// TwinCAT 3 PLC project TcLog
// Title: TcLog
// Company: Benedikt Geisler
// Author: Benedikt Geisler
// ProjectVersion: 0.6.1
// Description: TcLog provides logging functionality to TwinCAT.
// ProgramVersion: 3.1.4026.20
// libraries:
//   Tc2_Standard, * (Beckhoff Automation GmbH)
//   Tc2_System, * (Beckhoff Automation GmbH)
//   Tc2_Utilities, * (Beckhoff Automation GmbH)
//   Tc3_DynamicMemory, * (Beckhoff Automation GmbH)
// project tree:
//   / Constants.TcGVL (not stored)
//   Logger/Buffer/ LogEventRingBuffer.TcPOU, LogEventBuffer.TcIO
//   Logger/Functions/ DeviceIdentification.TcPOU, FindLastOccurrence.TcPOU, GetFileExtension.TcPOU, LogLevelToAdsLogMsgType.TcPOU, RollingIntervalDetector.TcPOU, ShortenInstancePath.TcPOU, SystemTimeToNlogString.TcPOU
//   Logger/DataTypes/ Error.TcDUT, ErrorCodes.TcDUT (not stored), LogEvent.TcDUT, LoggingConfiguration.TcDUT, LogLevel.TcDUT, RollingInterval.TcDUT
//   Logger/Formatters/ DefaultAdsLogEventFormatter.TcPOU, DefaultFileLogEventFormatter.TcPOU
//   Logger/Interfaces/ ILog.TcIO (not stored), ILogCore.TcIO, LogEventFormatter.TcIO
//   Logger/TargetAdapters/ AdsLogTargetAdapter.TcPOU, FileLogTargetAdapter.TcPOU, LogTargetAdapter.TcIO
//   Logger/ TcLog.TcPOU, TcLogCore.TcPOU, TcLogTrig.TcPOU
//   StringBuilder/Interfaces/ ILimitedStringBuilder.TcIO (not stored), IStringBuilder.TcIO
//   StringBuilder/ StringBuilder.TcPOU
//   Utils/ AnyToString.TcPOU, DateTime.TcPOU, DeleteOldFiles.TcPOU (not stored), DynamicStringBuffer.TcPOU, GetFileAgeInSeconds.TcPOU
//   Utils/DataTypes/ DeleteFilesState.TcDUT, PersistToFileState.TcDUT (not stored)

// ---- Logger/DataTypes/Error.TcDUT
/// This is the error type used in this library.
TYPE Error :
STRUCT
	Active : BOOL; // `TRUE` signals an active error
	Code : INT; // Error code of type `ErrorCodes`
	Info : Tc2_System.T_MaxString; // Plain text error message
END_STRUCT
END_TYPE

// ---- Logger/DataTypes/LogEvent.TcDUT
TYPE LogEvent :
STRUCT
	timestamp : Tc2_Utilities.TimeStruct;
	level : LogLevel;
	logger : T_MaxString;
	message : T_MaxString;
END_STRUCT
END_TYPE

// ---- Logger/DataTypes/LoggingConfiguration.TcDUT
/// Configuration of TcLogCore
TYPE LoggingConfiguration :
STRUCT
	/// Whether to include the instance path of TcLog into the log message or not.
	IncludeInstancePath : BOOL;
	
	/// What is the minimum log level that gets logged?
	MinimumLevel : LogLevel;
	
	/// Which delimiter should be used between the different parts of the log string?
	Delimiter : STRING(1);
	
	/// Format of timestamp. See `TcLogCore.TimestampFormat` for formatting options.
	TimestampFormat : STRING;
	
	/// Log only valid timestamps (skip log messages during time initialization (first few cycles)
	ValidTimestampsOnly: BOOL;
END_STRUCT
END_TYPE

// ---- Logger/DataTypes/LogLevel.TcDUT
/// Log level of message to be logged.
{attribute 'qualified_only'}
{attribute 'strict'}
{attribute 'to_string'}
TYPE LogLevel :
(
	Debug := 0,
	Information,
	Warning,
	Error,
	Fatal
);
END_TYPE

// ---- Logger/DataTypes/RollingInterval.TcDUT
/// Rolling interval to create a new log file when expired. 
{attribute 'qualified_only'}
{attribute 'strict'}
{attrivute 'to_string'}
TYPE RollingInterval :
(
	None := 0,
	Hourly,
	Daily,
	Weekly,
	Monthly,
	Yearly
);
END_TYPE

// ---- Utils/DataTypes/DeleteFilesState.TcDUT
// States for state machine used in `DeleteOldFiles`.
{attribute 'qualified_only'}
{attribute 'strict'}
TYPE INTERNAL DeleteFilesState :
(
	Idle := 0,
  SearchNextFile,
  WaitUntilExecutionDone,
  ProcessFoundFiles,
  CheckIfFileIsDirectory,
  CheckFileTime,
  DeleteFile,
  FileDeleted
);
END_TYPE

// ---- Logger/Buffer/LogEventBuffer.TcIO
INTERFACE PUBLIC LogEventBuffer EXTENDS __SYSTEM.IQueryInterface

{attribute 'monitoring':='call'}
PROPERTY PUBLIC IsFull : BOOL
GET
END_GET
END_PROPERTY

METHOD PUBLIC Pop : LogEvent
END_METHOD

METHOD PUBLIC Push : BOOL
VAR_INPUT
	event : LogEvent;
END_VAR
END_METHOD

{attribute 'monitoring':='call'}
PROPERTY PUBLIC Size : UDINT
GET
END_GET
END_PROPERTY

END_INTERFACE

// ---- Logger/Interfaces/ILogCore.TcIO
INTERFACE PUBLIC ILogCore EXTENDS __SYSTEM.IQueryInterface

// Logger method.
// Logs in the standard format. This includes
// - timestamp
// - log level
// - log message
// - instance path of logging source (optional)
// The message will only be logged if the logging level exceeds the configured minimum logging level.
METHOD PUBLIC LogStandardFormat : BOOL
VAR_INPUT
	instance_path : Tc2_System.T_MaxString; // Instance path of calling logger to locate source of logging message.
	level : LogLevel; // Log level of message.
	message : Tc2_System.T_MaxString; // Data to be logged. Additional formatting wil be done.
END_VAR
END_METHOD

END_INTERFACE

// ---- Logger/Interfaces/LogEventFormatter.TcIO
INTERFACE PUBLIC LogEventFormatter EXTENDS __SYSTEM.IQueryInterface

METHOD Format : T_MaxString
VAR_INPUT
	event : LogEvent;
END_VAR
END_METHOD

END_INTERFACE

// ---- Logger/TargetAdapters/LogTargetAdapter.TcIO
INTERFACE PUBLIC LogTargetAdapter EXTENDS __System.IQueryInterface

METHOD PUBLIC Run
END_METHOD

METHOD PUBLIC SendLogEvent : BOOL
VAR_INPUT
	event : LogEvent;
END_VAR
END_METHOD

END_INTERFACE

// ---- StringBuilder/Interfaces/IStringBuilder.TcIO
{attribute 'hide'}
INTERFACE INTERNAL IStringBuilder

METHOD Append : IStringBuilder // Append text TO t current build STRING.
VAR_INPUT
    Text : Tc2_System.T_MaxString; //Text to append to current build string
END_VAR
END_METHOD

METHOD AppendIf : IStringBuilder
VAR_INPUT
    Condition : BOOL;
    Text : Tc2_System.T_MaxString;
END_VAR
END_METHOD

METHOD InsertAtLocation : IStringBuilder
VAR_INPUT
    Text : Tc2_System.T_MaxString;
    Position : INT;
END_VAR
END_METHOD

METHOD PadLeft : IStringBuilder
VAR_INPUT
    text : Tc2_System.T_MaxString; // Text to append to current build string
    length : INT; // Total length of text + padding
    c : STRING(1); // Character to be padded left of text
END_VAR
END_METHOD

METHOD Reset : ILimitedStringBuilder //Reset current build STRING TO an empty STRING.
END_METHOD

METHOD ToString : Tc2_System.T_MaxString //Returns current build STRING.
END_METHOD

END_INTERFACE

// ---- Logger/Buffer/LogEventRingBuffer.TcPOU
FUNCTION_BLOCK PUBLIC LogEventRingBuffer
VAR_GENERIC CONSTANT
	capacity : UDINT := 100;
END_VAR
IMPLEMENTS LogEventBuffer
VAR
	buffer : ARRAY[0..capacity-1] OF LogEvent;
	head : UDINT;
	tail : UDINT;
	_size : UDINT;
END_VAR

{attribute 'monitoring':='call'}
PROPERTY PUBLIC IsFull : BOOL
GET // PUBLIC
IsFull := _size = capacity;
END_GET
END_PROPERTY

METHOD PUBLIC Pop : LogEvent
VAR
	item : LogEvent;
END_VAR
IF _size = 0 THEN
	RETURN;
END_IF

item := buffer[head];
buffer[head] := 0; // Help garbage collection
head := (head + 1) MOD capacity;
_size := _size - 1;
Pop := item;
END_METHOD

METHOD PUBLIC Push : BOOL
VAR_INPUT
	item : LogEvent;
END_VAR
buffer[tail] := item;
tail := (tail + 1) MOD capacity;
IF _size < capacity THEN
	_size := _size + 1;
ELSE
	head := (head + 1) MOD capacity; // Overwrite oldest element
END_IF
END_METHOD

{attribute 'monitoring':='call'}
PROPERTY PUBLIC Size : UDINT
GET // PUBLIC
Size := _size;
END_GET
END_PROPERTY

END_FUNCTION_BLOCK

// ---- Logger/Functions/DeviceIdentification.TcPOU
FUNCTION_BLOCK DeviceIdentification
VAR
	fb : FB_GetDeviceIdentificationEx;
	initialised : BOOL;
	
	is_windows : BOOL;
	is_windows_ce : BOOL;
	is_bsd : BOOL;
	is_linux : BOOL;
	
	path_delimiter : STRING(1);
END_VAR

METHOD PUBLIC Initialise : BOOL
VAR
	dev_id : Tc2_Utilities.ST_DeviceIdentificationEx;
END_VAR
IF initialised THEN
	Initialise := initialised;
	RETURN;
END_IF

fb(bExecute := TRUE);

IF NOT fb.bBusy THEN
	dev_id := fb.stDevIdent;
	initialised := TRUE;
	fb(bExecute := FALSE);
END_IF

IF Left(dev_id.strImageOsName, 10) = 'Windows CE' THEN
	is_windows_ce := TRUE;
ELSIF Left(dev_id.strImageOsName, 7) = 'Windows' THEN
	is_windows := TRUE; 
END_IF

IF is_windows OR is_windows_ce THEN
	path_delimiter := '\';
ELSE
	path_delimiter := '/';
END_IF
END_METHOD

{attribute 'monitoring':='call'}
PROPERTY PUBLIC IsBsd : BOOL
GET // PUBLIC
IsBsd := is_bsd;
END_GET
END_PROPERTY

{attribute 'monitoring':='call'}
PROPERTY PUBLIC IsLinux : BOOL
GET // PUBLIC
IsLinux := is_linux;
END_GET
END_PROPERTY

{attribute 'monitoring':='call'}
PROPERTY PUBLIC IsWindows : BOOL
GET // PUBLIC
IsWindows := is_windows;
END_GET
END_PROPERTY

{attribute 'monitoring':='call'}
PROPERTY PUBLIC IsWindowsCE : BOOL
GET // PUBLIC
IsWindowsCE := is_windows_ce;
END_GET
END_PROPERTY

{attribute 'monitoring':='call'}
PROPERTY PUBLIC PathDelimiter : STRING(1)
GET // PUBLIC
PathDelimiter := path_delimiter;
END_GET
END_PROPERTY

END_FUNCTION_BLOCK

// ---- Logger/Functions/FindLastOccurrence.TcPOU
FUNCTION FindLastOccurrence : INT
VAR_INPUT
	within_text : T_MaxString;
	find_text : T_MaxString; 
END_VAR
VAR
	complete : BOOL;
	found_index : INT;
	new_within_text : T_MaxString;
	new_found_index : INT;
END_VAR

new_within_text := within_text;

REPEAT
	new_found_index := Find(new_within_text, find_text);
	
	IF new_found_index <> 0 THEN
		found_index := found_index + new_found_index;
		new_within_text := Right(new_within_text, Len(new_within_text) - new_found_index);
	ELSE
		complete := TRUE;
	END_IF
UNTIL complete
END_REPEAT;

FindLastOccurrence := found_index;

END_FUNCTION

// ---- Logger/Functions/GetFileExtension.TcPOU
FUNCTION GetFileExtension : T_MaxString
VAR_INPUT
	file_name : T_MaxString;
END_VAR
VAR
	last_separator_index : INT;
	extension : T_MaxString;
END_VAR

last_separator_index := FindLastOccurrence(file_name, '.');
extension := SEL(last_separator_index <> 0, '', Right(file_name, Len(file_name) - last_separator_index));
GetFileExtension := extension;

END_FUNCTION

// ---- Logger/Functions/LogLevelToAdsLogMsgType.TcPOU
// Converts TcLog.LogLevels into Tc2_System.AdsLog_MsgType.
//{attribute 'hide'}
FUNCTION INTERNAL LogLevelToAdsLogMsgType : DWORD
VAR_INPUT
  level : LogLevel;
END_VAR

CASE level OF
	LogLevel.Debug,
	LogLevel.Information:
		LogLevelToAdsLogMsgType := Tc2_System.AdsLog_MsgType_Hint;
		
	LogLevel.Warning:
		LogLevelToAdsLogMsgType := Tc2_System.AdsLog_MsgType_Warn;
		
	LogLevel.Error,
	LogLevel.Fatal:
		LogLevelToAdsLogMsgType := Tc2_System.AdsLog_MsgType_Error;
ELSE
	LogLevelToAdsLogMsgType := Tc2_System.AdsLog_MsgType_Hint;
END_CASE

END_FUNCTION

// ---- Logger/Formatters/DefaultAdsLogEventFormatter.TcPOU
{attribute 'linkalways'}
{attribute 'no_explicit_call' := 'This FB is a CLASS and must be accessed using methods or properties'}
FUNCTION_BLOCK DefaultAdsLogEventFormatter IMPLEMENTS LogEventFormatter
VAR
END_VAR

METHOD PUBLIC Format : T_MaxString
VAR_INPUT
	event : LogEvent;
END_VAR
VAR_INST
	{attribute 'hide'}
	message_builder : StringBuilder;
END_VAR
VAR CONSTANT
	DELIMITER : STRING := '|';
END_VAR
Format := message_builder
	.Reset()
	.Append(event.logger)
	.Append(DELIMITER)
	.Append(event.message)
	.ToString();
END_METHOD

END_FUNCTION_BLOCK

// ---- StringBuilder/StringBuilder.TcPOU
FUNCTION_BLOCK INTERNAL StringBuilder IMPLEMENTS IStringBuilder, ILimitedStringBuilder
VAR
  {attribute 'hide'}
  _workString : Tc2_System.T_MaxString;
END_VAR

METHOD PUBLIC Append : IStringBuilder // Append text TO t current build STRING.
VAR_INPUT
  text : Tc2_System.T_MaxString; //text to append to current build string
END_VAR
_workString:= Tc2_Standard.CONCAT(_workString,text);
Append := THIS^;
END_METHOD

METHOD PUBLIC AppendIf : IStringBuilder
VAR_INPUT
  condition : BOOL;
  text : Tc2_System.T_MaxString;
END_VAR
IF condition THEN
  _workString:= Tc2_Standard.CONCAT(_workString,text);
END_IF
AppendIf := THIS^;
END_METHOD

METHOD PUBLIC InsertAtLocation : IStringBuilder
VAR_INPUT
  text : Tc2_System.T_MaxString;
  position : INT;
END_VAR
_workString := Tc2_Standard.INSERT(_workSTring,text,position);
InsertAtLocation  := THIS^;
END_METHOD

METHOD PadLeft : IStringBuilder
VAR_INPUT
  text : Tc2_System.T_MaxString; // Text to append to current build string
  length : INT; // Total length of text + padding
  c : STRING(1); // Character to be padded left of text
END_VAR
VAR
  i : INT;
  padLength : INT;
END_VAR
// Add left padding
padLength := Tc2_Standard.LEN(text) - length;
FOR i := 1 TO padLength DO
  _workString:= Tc2_Standard.CONCAT(_workString, c);
END_FOR

// Add text
_workString:= Tc2_Standard.CONCAT(_workString,text);

PadLeft := THIS^;
END_METHOD

METHOD PUBLIC Reset : ILimitedStringBuilder //Reset current build STRING TO an empty STRING.
_workString:='';
Reset := THIS^;
END_METHOD

METHOD PUBLIC ToString : Tc2_System.T_MaxString //Returns current build STRING.
ToString := _workString;
END_METHOD

END_FUNCTION_BLOCK

// ---- Logger/Formatters/DefaultFileLogEventFormatter.TcPOU
{attribute 'linkalways'}
{attribute 'no_explicit_call' := 'This FB is a CLASS and must be accessed using methods or properties'}
FUNCTION_BLOCK DefaultFileLogEventFormatter IMPLEMENTS LogEventFormatter
VAR
END_VAR

METHOD PUBLIC Format : T_MaxString
VAR_INPUT
	event : LogEvent;
END_VAR
VAR_INST
	{attribute 'hide'}
	message_builder : StringBuilder;
END_VAR
VAR CONSTANT
	DELIMITER : STRING := '|';
END_VAR
Format := message_builder
	.Reset()
	.Append(SystemTimeToNlogString(event.timestamp))
	.Append(DELIMITER)
	.Append(TO_STRING(event.level))
	.Append(DELIMITER)
	.Append(event.logger)
	.Append(DELIMITER)
	.Append(event.message)
	.ToString();
END_METHOD

END_FUNCTION_BLOCK

// ---- Logger/Functions/SystemTimeToNlogString.TcPOU
FUNCTION INTERNAL SystemTimeToNlogString : T_MaxString
VAR_INPUT
	system_time : Tc2_Utilities.TimeStruct;
END_VAR

SystemTimeToNlogString := Tc2_Standard.Replace(Tc2_Utilities.SystemTime_To_String(system_time), ' ', 1, 11);

END_FUNCTION

// ---- Logger/Functions/RollingIntervalDetector.TcPOU
{attribute 'linkalways'}
{attribute 'no_explicit_call' := 'This FB is a CLASS and must be accessed using methods or properties'}
FUNCTION_BLOCK PUBLIC RollingIntervalDetector
VAR
	new_hour : Tc2_Standard.R_Trig;
	new_day : Tc2_Standard.R_Trig;
	new_week : Tc2_Standard.R_Trig;
	new_month : Tc2_Standard.R_Trig;
	new_year : Tc2_Standard.R_Trig;
	
	hour_rolled : BOOL;
	day_rolled : BOOL;
	week_rolled : BOOL;
	month_rolled : BOOL;
	year_rolled : BOOL;
END_VAR

PROPERTY PUBLIC DayRolled : BOOL
GET // PUBLIC
END_GET
END_PROPERTY

PROPERTY PUBLIC HourRolled : BOOL
GET // PUBLIC
END_GET
END_PROPERTY

METHOD PUBLIC IntervalRolled : BOOL
VAR_INPUT
	rolling_interval : RollingInterval;
END_VAR
CASE rolling_interval OF
	RollingInterval.Hourly:
		IntervalRolled := HourRolled;
		
	RollingInterval.Daily:
		IntervalRolled := DayRolled;
		
	RollingInterval.Weekly:
		IntervalRolled := WeekRolled;
		
	RollingInterval.Monthly:
		IntervalRolled := MonthRolled;
		
	RollingInterval.Yearly:
		IntervalRolled := YearRolled;
END_CASE
END_METHOD

PROPERTY PUBLIC MonthRolled : BOOL
GET // PUBLIC
END_GET
END_PROPERTY

METHOD PUBLIC Run
VAR_INPUT
	current_utc_time : Tc2_Utilities.TimeStruct;
END_VAR
new_hour(
	Clk := (current_utc_time.wMinute = 0 AND current_utc_time.wSecond = 0), 
	Q => hour_rolled
);

new_day(
	Clk := (hour_rolled AND current_utc_time.wHour = 0), 
	Q => day_rolled
);

new_week(
	Clk := (day_rolled AND current_utc_time.wDayOfWeek = 0),
	Q => week_rolled
);

new_month(
	Clk := (day_rolled AND current_utc_time.wDay = 1),
	Q => month_rolled
);

new_year(
	Clk := (day_rolled AND current_utc_time.wMonth = 1 AND current_utc_time.wDay = 1),
	Q => year_rolled
);
END_METHOD

PROPERTY PUBLIC WeekRolled : BOOL
GET // PUBLIC
END_GET
END_PROPERTY

PROPERTY PUBLIC YearRolled : BOOL
GET // PUBLIC
END_GET
END_PROPERTY

END_FUNCTION_BLOCK

// ---- Logger/Functions/ShortenInstancePath.TcPOU
FUNCTION INTERNAL ShortenInstancePath : T_MaxString
VAR_INPUT
	path : Tc2_System.T_MaxString; // Instance path to be shortened.
END_VAR
VAR
	i : UINT;
	shortened_path : Tc2_System.T_MaxString;
	position_in_string : INT := 0;
	position_of_last_dot : INT := 0;
END_VAR

shortened_path := path;

// Find last '.'
WHILE(Tc2_Standard.FIND(shortened_path, '.') > 0) DO
	position_in_string := Tc2_Standard.Find(shortened_path, '.');
	shortened_path := Tc2_Standard.Delete(shortened_path, position_in_string + 1, 0); 
	position_of_last_dot := position_of_last_dot + position_in_string;
END_WHILE

shortened_path := Path;

// Delete instantiation of this FB (obvious information)
shortened_path := Tc2_Standard.Delete(shortened_path, Tc2_Standard.Len(shortened_path) - position_of_last_dot + 1, position_of_last_dot);

// Delete project information
position_in_string := Tc2_Standard.Find(shortened_path, '.');
shortened_path := Tc2_Standard.Delete(shortened_path, position_in_string + 1, 0);

// Delete PLC information
position_in_string := Tc2_Standard.Find(shortened_path, '.');
shortened_path := Tc2_Standard.Delete(shortened_path, position_in_string + 1, 0);

ShortenInstancePath := shortened_path;

END_FUNCTION

// ---- Logger/TargetAdapters/AdsLogTargetAdapter.TcPOU
{attribute 'linkalways'}
{attribute 'no_explicit_call' := 'This FB is a CLASS and must be accessed using methods or properties'}
FUNCTION_BLOCK PUBLIC AdsLogTargetAdapter IMPLEMENTS LogTargetAdapter
VAR
	formatter : DefaultAdsLogEventFormatter;
END_VAR

METHOD PUBLIC Run
// Do nothing for this, as it directly logs
END_METHOD

METHOD PUBLIC SendLogEvent : BOOL
VAR_INPUT
	event : LogEvent;
END_VAR
Tc2_System.AdsLogStr(
	AdsLog_MsgType_Log OR LogLevelToAdsLogMsgType(event.level), 
	formatter.Format(event), 
	''
);
END_METHOD

END_FUNCTION_BLOCK

// ---- Logger/TargetAdapters/FileLogTargetAdapter.TcPOU
{attribute 'linkalways'}
{attribute 'no_explicit_call' := 'This FB is a CLASS and must be accessed using methods or properties'}
FUNCTION_BLOCK PUBLIC FileLogTargetAdapter IMPLEMENTS LogTargetAdapter
VAR CONSTANT
	message_buffer_capacity : UDINT := 100; // Number of messages that can be buffered
END_VAR
VAR
	// Configuration
	file_path : STRING := 'C:\';
	file_name : STRING := 'tclog.log';
	
	rolling_interval : RollingInterval := RollingInterval.Daily;
	/// When should old log files be deleted? Unit: days. Set it to `0` if log files should never be deleted. 
	log_lifespan : UINT := 0;
	timestamp_format : STRING := 'YYYYMMDD_hhmm_';

	log_cache : DynamicStringBuffer;
	date_time : DateTime;

	utc_time_as_file_time : Tc2_Utilities.T_FileTime; // Current utc time as filetime
	local_time_as_system_time : Tc2_Utilities.TimeStruct; // Current local time as timestring
	local_time_as_string : STRING; // Current local time as string

	formatter : DefaultFileLogEventFormatter;

	_error : Error; // Contains information about internal error.
	_busy : BOOL; // Logger is busy, typically with writing logs to the file system.
	
	rolling_interval_detector : RollingIntervalDetector;
	
	file_name_truncated : STRING;
	file_name_extension : STRING;
END_VAR

/// Configuration method which sets the lifespan of log files. Once exceeded, they will be deleted.
METHOD PUBLIC DeleteLogFilesAfterDays : REFERENCE TO FileLogTargetAdapter
VAR_INPUT
	/// Lifespan of logfiles in days.
	lifespan : UINT; 
END_VAR
log_lifespan := lifespan;

DeleteLogFilesAfterDays REF= THIS^;
END_METHOD

//FB_Init is always available implicitly and it is used primarily for initialization.
//The return value is not evaluated. For a specific influence, you can also declare the
//methods explicitly and provide additional code there with the standard initialization
//code. You can evaluate the return value.
METHOD FB_Init: BOOL
VAR_INPUT
    bInitRetains: BOOL; // TRUE: the retain variables are initialized (reset warm / reset cold)
    bInCopyCode: BOOL;  // TRUE: the instance will be copied to the copy code afterward (online change)   
END_VAR
log_cache.Init(message_buffer_capacity * (Tc2_System.Max_String_Length + Constants.FifoOverhead));
END_METHOD

/// Configuration method
/// Sets file_name of log file.
METHOD PUBLIC FileName : REFERENCE TO FileLogTargetAdapter
VAR_INPUT
	/// File name where the logs should be written to. Should not include path.
	file_name : STRING;
END_VAR
VAR
	last_period_index : INT;
END_VAR
THIS^.file_name := file_name;

last_period_index := FindLastOccurrence(file_name, '.');

IF last_period_index <> 0 THEN
	file_name_extension := GetFileExtension(file_name);
ELSE
	file_name_extension := 'log';
END_IF

FileName REF= THIS^;
END_METHOD

/// Configuration method
/// Sets file_path for log files.
METHOD PUBLIC FilePath : REFERENCE TO FileLogTargetAdapter
VAR_INPUT
	/// File path where the logs should be written to. Will be prefixed to `FileName`
	file_path : STRING; 
END_VAR
THIS^.file_path := file_path;

FilePath REF= THIS^;
END_METHOD

/// Flushes the logging cache. All messages that have not yet been processed will be lost.
METHOD PUBLIC FlushCache : BOOL
log_cache.FlushCache();
END_METHOD

METHOD PUBLIC Run
VAR_INST
	new_day : Tc2_Standard.R_Trig; 
	delete_expired_log_files : DeleteOldFiles;
	file_name_string_builder : StringBuilder;
	time_stamp : STRING; // Timestamp used for filename
	time_info_ready : BOOL := FALSE; // Set to true once the time information is available
	internal_error_occured : BOOL; // Aux variable to log internal errors to Error-property.
END_VAR
// Generate time data (shared state)
date_time.CyclicCall();
IF date_time.Done THEN
	time_info_ready := TRUE;
END_IF

local_time_as_system_time := date_time.AsLocalSystemTime;
local_time_as_string := date_time.AsLocalSystemTimeString;
utc_time_as_file_time := date_time.AsUtcFileTime;

rolling_interval_detector.Run(local_time_as_system_time);

// Generate new timestamp for filename
IF rolling_interval_detector.IntervalRolled(rolling_interval) OR date_time.Done THEN
	time_stamp := date_time.ToFormatString(timestamp_format);
END_IF

// Delete expired log files
new_day(Clk := local_time_as_system_time.wHour = 0);
delete_expired_log_files(
	StartScan 			:= 	new_day.Q AND (log_lifespan > 0),
	ExpirationInDays 	:=	log_lifespan,
	FilePath			:=	file_path,
	FileName 			:=	file_name,
	CurrentUtcTime 		:= 	utc_time_as_file_time	
);
IF delete_expired_log_files.Error.Active THEN
	internal_error_occured := TRUE;
	_error := delete_expired_log_files.Error;
END_IF
		
// Persist logging messages to file
log_cache.PersistToFile(
	time_info_ready,
	file_name_string_builder
		.Reset()
		.Append(file_path)
		.AppendIf(Tc2_Standard.Right(file_path, 1) <> '\', '\')
		.Append(time_stamp)
		.Append(file_name)
		.ToString()
);
IF log_cache.Error.Active THEN
	internal_error_occured := TRUE;
	_error := log_cache.Error;
END_IF

// Reset error flag each cycle to automatically confirm errors once they are gone.
IF NOT internal_error_occured THEN
	_error.Active := FALSE;
	_error.Code := ErrorCodes.None;
	_error.Info := '';
END_IF
internal_error_occured := FALSE;
END_METHOD

METHOD PUBLIC SendLogEvent : BOOL
VAR_INPUT
	event : LogEvent;
END_VAR
log_cache.AddLine(formatter.Format(event));
END_METHOD

/// Configuration method.
/// Sets the rolling interval of the log file. Once the rolling interval
/// expires, a file name with a new timestamp will be generated.
METHOD PUBLIC SetRollingInterval : REFERENCE TO FileLogTargetAdapter
VAR_INPUT
	/// Rolling interval for log file. Once exceeded, a new log file will be created.
	interval : RollingInterval; 
END_VAR
rolling_interval := interval;

SetRollingInterval REF= THIS^;
END_METHOD

END_FUNCTION_BLOCK

// ---- Logger/TcLog.TcPOU
/// `TcLog` is the client side of the logger.  
///
/// It is used to send the logs to `TcLogCore`. Typically, it is instantiated
/// once in each `FUNCTION_BLOCK` or `PROGRAM` where logging is done. The same 
/// instance can then be used for all logging within that POU. 
///
/// `TcLog` implements a string builder that facilitates the compilation of the log
/// message without the need for external data type conversions or multiple chained `CONCAT` calls.
/// See the method section for more information.
///
/// The last method to call after the log message has been built is one of ´[Debug|Information|Warning|Error|Fatal]`. 
/// This sets the log level of the message and sends it off to the log message queue of `TcLogCore` where it will
/// be processed according to its configuration.
{attribute 'linkalways'}
{attribute 'no_explicit_call' := 'This FB is a CLASS and must be accessed using methods or properties'}
//{attribute 'hide_all_locals'}
{attribute 'reflection'} 
FUNCTION_BLOCK PUBLIC TcLog IMPLEMENTS ILog
VAR
	log_condition_satisfied : BOOL; // flag that indicates, whether log condition has been satisfied.
								    // Logging will only be carried out it this evaluates to TRUE.                    
	
	log_data_initialised : BOOL; // flag that indicate, whether log data has been initialized.
							     // Necessary for configuration methods to provide a fluent interface.                            
	
	log_data : Tc2_System.T_MaxString; // contains message to be logged.
	used_logger : ILogCore;
	
	{attribute 'instance-path'} 
	{attribute 'noinit'} 
	instance_path : STRING; // contains instance path
END_VAR
VAR_STAT
	{attribute 'hide'}
	logger_singleton_instance : ILogCore; // Wires up TcLog ("Client") to TcLogCore ("Server") (Singleton-Behaviour)
END_VAR
VAR CONSTANT
	INVALID_LOGGER_REFERENCE : UDINT := 0;
END_VAR

/// Appends any given data to the log string. The type of the provided data
/// has to be one of the [standard data types](https://infosys.beckhoff.com/english.php?content=../content/1033/tc3_plc_intro/2529388939.html&id=).
/// This method can be chained.
METHOD AppendAny : REFERENCE TO TcLog
VAR_INPUT
	/// data to be appended to log string.
	data : ANY;
END_VAR
InitializeLogData();

log_data := Tc2_Standard.CONCAT(log_data, AnyToString(data));

AppendAny REF= THIS^;
END_METHOD

/// Appends a BYTE to the log string.
/// This method can be chained.
METHOD PUBLIC AppendByte : REFERENCE TO TcLog
VAR_INPUT
	/// data to be appended to log string.
	data : BYTE;
END_VAR
AppendByte REF= AppendString(TO_STRING(data));
END_METHOD

/// Appends a DATE to the log string.
/// This method can be chained.
METHOD PUBLIC AppendDate : REFERENCE TO TcLog
VAR_INPUT
  /// data to be appended to log string.
  data : DATE;
END_VAR
AppendDate REF= AppendString(TO_STRING(data));
END_METHOD

/// Appends a DATE_AND_TIME to the log string.
/// This method can be chained.
METHOD PUBLIC AppendDateAndTime : REFERENCE TO TcLog
VAR_INPUT
  /// data to be appended to log string.
  data : DATE_AND_TIME;
END_VAR
AppendDateAndTime REF= AppendString(TO_STRING(data));
END_METHOD

/// Appends a DINT to the log string.
/// This method can be chained.
METHOD PUBLIC AppendDint : REFERENCE TO TcLog
VAR_INPUT
	/// data to be appended to log string.
	data : DINT;
END_VAR
AppendDint REF= AppendString(TO_STRING(data));
END_METHOD

/// Appends a DWORD to the log string.
/// This method can be chained.
METHOD PUBLIC AppendDword : REFERENCE TO TcLog
VAR_INPUT
  /// data to be appended to log string.
  data : DWORD;
END_VAR
AppendDword REF= AppendString(TO_STRING(data));
END_METHOD

/// Appends an INT to the log string.
/// This method can be chained.
METHOD PUBLIC AppendInt : REFERENCE TO TcLog
VAR_INPUT
  /// data to be appended to log string.
  data : INT;
END_VAR
AppendInt REF= AppendString(TO_STRING(data));
END_METHOD

/// Appends a LDATE to the log string.
/// This method can be chained.
METHOD PUBLIC AppendLDate : REFERENCE TO TcLog
VAR_INPUT
  /// data to be appended to log string.
  data : LDATE;
END_VAR
AppendLDate REF= AppendString(TO_STRING(data));
END_METHOD

/// Appends a LDATE_AND_TIME to the log string.
/// This method can be chained.
METHOD PUBLIC AppendLDateAndTime : REFERENCE TO TcLog
VAR_INPUT
  /// data to be appended to log string.
  data : LDATE_AND_TIME;
END_VAR
AppendLDateAndTime REF= AppendString(TO_STRING(data));
END_METHOD

/// Appends an LINT to the log string.
/// This method can be chained.
METHOD PUBLIC AppendLint : REFERENCE TO TcLog
VAR_INPUT
  /// data to be appended to log string.
  data : LINT;
END_VAR
AppendLint REF= AppendString(TO_STRING(data));
END_METHOD

/// Appends an LREAL to the log string.
/// This method can be chained.
METHOD PUBLIC AppendLreal : REFERENCE TO TcLog
VAR_INPUT
  /// data to be appended to log string.
  data : LREAL;
END_VAR
AppendLreal REF= AppendString(TO_STRING(data));
END_METHOD

/// Appends a LTIME_OF_DAY to the log string.
/// This method can be chained.
METHOD PUBLIC AppendLTimeOfDay : REFERENCE TO TcLog
VAR_INPUT
  /// data to be appended to log string.
  data : LTIME_OF_DAY;
END_VAR
AppendLTimeOfDay REF= AppendString(TO_STRING(data));
END_METHOD

/// Appends an LWORD to the log string.
/// This method can be chained.
METHOD PUBLIC AppendLword : REFERENCE TO TcLog
VAR_INPUT
  /// data to be appended to log string.
  data : LWORD;
END_VAR
AppendLword REF= AppendString(TO_STRING(data));
END_METHOD

/// Appends a REAL to the log string.
/// This method can be chained.
METHOD PUBLIC AppendReal : REFERENCE TO TcLog
VAR_INPUT
  /// data to be appended to log string.
  data : REAL;
END_VAR
AppendReal REF= AppendString(TO_STRING(data));
END_METHOD

/// Appends a SINT to the log string.
/// This method can be chained.
METHOD PUBLIC AppendSint : REFERENCE TO TcLog
VAR_INPUT
  /// data to be appended to log string.
  data : SINT;
END_VAR
AppendSint REF= AppendString(TO_STRING(data));
END_METHOD

/// Appends another string to the log message.
/// This method can be chained.
METHOD AppendString : REFERENCE TO TcLog
VAR_INPUT
	/// data to be appended to log string.
	data : Tc2_System.T_MaxString; 
END_VAR
InitializeLogData();

log_data := Tc2_Standard.CONCAT(log_data, data);
  
AppendString REF= THIS^;
END_METHOD

/// Appends a TIME_OF_DAY to the log string.
/// This method can be chained.
METHOD PUBLIC AppendTimeOfDay : REFERENCE TO TcLog
VAR_INPUT
  /// data to be appended to log string.
  data : TIME_OF_DAY;
END_VAR
AppendTimeOfDay REF= AppendString(TO_STRING(data));
END_METHOD

/// Appends a UDINT to the log string.
/// This method can be chained.
METHOD PUBLIC AppendUdint : REFERENCE TO TcLog
VAR_INPUT
  /// data to be appended to log string.
  data : UDINT;
END_VAR
AppendUdint REF= AppendString(TO_STRING(data));
END_METHOD

/// Appends a UINT to the log string.
/// This method can be chained.
METHOD PUBLIC AppendUint : REFERENCE TO TcLog
VAR_INPUT
  /// data to be appended to log string.
  data : UINT;
END_VAR
AppendUint REF= AppendString(TO_STRING(data));
END_METHOD

/// Appends a ULINT to the log string.
/// This method can be chained.
METHOD PUBLIC AppendUlint : REFERENCE TO TcLog
VAR_INPUT
  /// data to be appended to log string.
  data : ULINT;
END_VAR
AppendUlint REF= AppendString(TO_STRING(data));
END_METHOD

/// Appends a USINT to the log string.
/// This method can be chained.
METHOD PUBLIC AppendUsint : REFERENCE TO TcLog
VAR_INPUT
  /// data to be appended to log string.
  data : USINT;
END_VAR
AppendUsint REF= AppendString(TO_STRING(data));
END_METHOD

/// Appends information about the given variable to the log string. 
/// This method can be chained.
/// Example: 

/// ```st
/// VAR
///   Logger: TcLog;
///    myInt : INT := 10;
///   myVarInfo : __SYSTEM.VAR_INFO := __VARINFO(myInt);
/// END_VAR
/// Logger.AppendVariable(myVarInfo, myInt);
/// ```
///
METHOD AppendVariable : REFERENCE TO TcLog
VAR_INPUT
	/// [VAR_INFO](https://infosys.beckhoff.com/index.php?content=../content/1031/tc3_plc_intro/3527777675.html&id=) of variable to be appended to log string.
	varInfo : __SYSTEM.VAR_INFO;
	/// Value of variable to be appended to log string.
	value : ANY; 
END_VAR
VAR
	format : Tc2_Utilities.FB_FormatString;
	symbolName : Tc2_System.T_MaxString;
	typeName : Tc2_System.T_MaxString;
END_VAR
InitializeLogData();

symbolName := varInfo.Symbol;
typeName := varInfo.TypeName; 

format(
  sFormat := '%s [%s] : ',
  arg1 := Tc2_Utilities.F_String(symbolName),
  arg2 := Tc2_Utilities.F_String(typeName));
  
AppendString(format.sOut);
AppendAny(value);

AppendVariable REF= THIS^;
END_METHOD

/// Appends a WORD to the log string.
/// This method can be chained.
METHOD PUBLIC AppendWord : REFERENCE TO TcLog
VAR_INPUT
  /// data to be appended to log string.
  data : WORD;
END_VAR
AppendWord REF= AppendString(TO_STRING(data));
END_METHOD

/// Logs the log string in DEBUG level.
METHOD PUBLIC Debug : BOOL
VAR_INPUT
	/// Message to be appended to log string.
	message : Tc2_System.T_MaxString; 
END_VAR
LogWithLevel(message, LogLevel.Debug);
END_METHOD

/// Logs the log string in ERROR level.
METHOD PUBLIC Error
VAR_INPUT
	/// Message to be appended to log string.
	message : Tc2_System.T_MaxString; 
END_VAR
LogWithLevel(message, LogLevel.Error);
END_METHOD

/// Logs the log string in FATAL level.
METHOD PUBLIC Fatal : BOOL
VAR_INPUT
	/// Message to be appended to log string.
	message : Tc2_System.T_MaxString; 
END_VAR
LogWithLevel(message, LogLevel.Fatal);
END_METHOD

/// Logs the log string in INFORMATION level.
METHOD PUBLIC Information : BOOL
VAR_INPUT
	/// Message to be appended to log string.
	message : Tc2_System.T_MaxString; 
END_VAR
LogWithLevel(message, LogLevel.Information);
END_METHOD

/// Initializes the reference to the core logger. Should only be called once from the core logger directly.
METHOD PUBLIC Init : BOOL
VAR_INPUT
	/// Reference to TcLoggerCore instance.
	log_core : ILogCore; 
END_VAR
IF logger_singleton_instance = 0 THEN
	logger_singleton_instance := log_core;
END_IF
END_METHOD

// Necessary to provide a fluent interface of the function. 
// Has to be called at the begin of any method that returns a reference to THIS^
METHOD PRIVATE InitializeLogData : BOOL
IF NOT log_data_initialised THEN
	log_condition_satisfied := TRUE;
	log_data := '';
	log_data_initialised := TRUE;
	
	IF used_logger = 0 THEN
		used_logger := logger_singleton_instance;
	END_IF
END_IF
END_METHOD

METHOD PUBLIC LogWithLevel
VAR_INPUT
	message : Tc2_System.T_MaxString;
	level : LogLevel;
END_VAR
VAR
	shortened_instance_path : T_MaxString;
	modified_message : T_MaxString;
END_VAR
InitializeLogData();

IF log_condition_satisfied THEN
	IF used_logger <> INVALID_LOGGER_REFERENCE THEN
		modified_message := Tc2_Standard.Concat(log_data, message);
 		shortened_instance_path := ShortenInstancePath(instance_path);
		used_logger.LogStandardFormat(
			shortened_instance_path,
			level,
			modified_message
		);
	ELSE
		Tc2_System.AdsLogStr(
			AdsLog_MsgType_Log OR LogLevelToAdsLogMsgType(LogLevel.Error),
			'used_logger: No valid reference',
			''
		); 
	END_IF
END_IF

log_data_initialised := FALSE;
END_METHOD

/// Conditional execution of the log command. Only executes logging when Cond = TRUE.
METHOD PUBLIC OnCondition : REFERENCE TO TcLog
VAR_INPUT
  /// Logs data only if this condition evaluates to TRUE.
  cond : BOOL; 
END_VAR
InitializeLogData();

log_condition_satisfied := cond;

OnCondition REF= THIS^;
END_METHOD

/// Initializes the reference to the core logger. This enables you to use several
/// loggers with different configurations in one project.
METHOD PUBLIC SetLogger : BOOL
VAR_INPUT
  /// Reference to Core Logger
  ref2Core : ILogCore; 
END_VAR
used_logger := ref2Core;
END_METHOD

/// Logs directly to ADS log, ignoring the settings of the base logger.
METHOD PUBLIC ToAdsLog : BOOL
VAR_INPUT
  /// Log level in which message should be logged to ADS.
  level : LogLevel; 
END_VAR
InitializeLogData();

IF log_condition_satisfied THEN
	Tc2_System.AdsLogStr(
		AdsLog_MsgType_Log OR LogLevelToAdsLogMsgType(level),
		log_data,
		''
	); 
END_IF

log_data_initialised := FALSE;
END_METHOD

/// Logs the log string in WARNING level.
METHOD PUBLIC Warning
VAR_INPUT
	/// Message to be appended to log string.
	message : Tc2_System.T_MaxString; 
END_VAR
LogWithLevel(message, LogLevel.Warning);
END_METHOD

END_FUNCTION_BLOCK

// ---- Utils/AnyToString.TcPOU
/// Converts value of input data to string, where the input type can be any of 
/// the standard data types.
FUNCTION AnyToString : Tc2_System.T_MaxString
VAR_INPUT
	/// Input data
	data : ANY;
END_VAR
VAR
	any_byte : POINTER TO BYTE;
	any_usint : POINTER TO USINT;
	_any_int : POINTER TO INT;
	any_uint : POINTER TO UINT;
	any_udint : POINTER TO UDINT;
	_anySInt : POINTER TO SINT;
	_anyDInt : POINTER TO DINT;
	_anyLInt : POINTER TO LINT;
	_anyULInt : POINTER TO ULINT;
	_anyWord : POINTER TO WORD;
	_anyLWord : POINTER TO LWORD;
	_anyReal : POINTER TO REAL;
	_anyLReal : POINTER TO LREAL;
	_anyDateAndTime : POINTER TO DATE_AND_TIME;
	_anyDate : POINTER TO DATE;
	_anyTime : POINTER TO TIME;
	_anyWString : POINTER TO WSTRING;
	_anyTOD : POINTER TO TOD;
	_anyString : POINTER TO STRING;
	_string : T_MAXSTRING;
	_wString : WSTRING;
END_VAR

IF data.TypeClass = __SYSTEM.TYPE_CLASS.TYPE_BYTE THEN
  any_byte := data.pValue;
  AnyToString := BYTE_TO_STRING(any_byte^);
    
ELSIF data.TypeClass = __SYSTEM.TYPE_CLASS.TYPE_INT THEN
  _any_int := data.pValue;
  AnyToString := INT_TO_STRING(_any_int^);
    
ELSIF data.TypeClass = __SYSTEM.TYPE_CLASS.TYPE_UINT THEN
  any_uint := data.pValue;
  AnyToString := UINT_TO_STRING(any_uint^);
    
ELSIF data.TypeClass = __SYSTEM.TYPE_CLASS.TYPE_UDINT THEN
  any_udint := data.pValue;
  AnyToString := UDINT_TO_STRING(any_udint^);
    
ELSIF data.TypeClass = __SYSTEM.TYPE_CLASS.TYPE_SINT THEN
  _anySInt := data.pValue;
  AnyToString := SINT_TO_STRING(_anySInt^);
    
ELSIF data.TypeClass = __SYSTEM.TYPE_CLASS.TYPE_USINT THEN
  any_usint := data.pValue;
  AnyToString := USINT_TO_STRING(any_usint^);
    
ELSIF data.TypeClass = __SYSTEM.TYPE_CLASS.TYPE_DINT THEN
  _anyDInt := data.pValue;
  AnyToString := DINT_TO_STRING(_anyDInt^);
    
ELSIF data.TypeClass = __SYSTEM.TYPE_CLASS.TYPE_LINT THEN
  _anyLInt := data.pValue;
  AnyToString := LINT_TO_STRING(_anyLInt^);
      
ELSIF data.TypeClass = __SYSTEM.TYPE_CLASS.TYPE_ULINT THEN
  _anyULInt := data.pValue;
  AnyToString := ULINT_TO_STRING(_anyULInt^);
  
ELSIF data.TypeClass = __SYSTEM.TYPE_CLASS.TYPE_WORD THEN
  _anyWord := data.pValue;
  AnyToString := WORD_TO_STRING(_anyWord^);
    
ELSIF data.TypeClass = __SYSTEM.TYPE_CLASS.TYPE_LWORD THEN
  _anyLWord := data.pValue;
  AnyToString := LWORD_TO_STRING(_anyLWord^);
  
ELSIF data.TypeClass = __SYSTEM.TYPE_CLASS.TYPE_REAL THEN
  _anyReal := data.pValue;
  AnyToString := REAL_TO_STRING(_anyReal^);
  
ELSIF data.TypeClass = __SYSTEM.TYPE_CLASS.TYPE_LREAL THEN
  _anyLReal := data.pValue;
  AnyToString := LREAL_TO_STRING(_anyLReal^);
  
ELSIF data.TypeClass = __SYSTEM.TYPE_CLASS.TYPE_DATEANDTIME THEN
  _anyDateAndTime := data.pValue;
  AnyToString := DT_TO_STRING(_anyDateAndTime^);  
  
ELSIF data.TypeClass = __SYSTEM.TYPE_CLASS.TYPE_DATE THEN
  _anyDate := data.pValue;
  AnyToString := DATE_TO_STRING(_anyDate^);
  
ELSIF data.TypeClass = __SYSTEM.TYPE_CLASS.TYPE_TIME THEN
  _anyTime := data.pValue;
  AnyToString := TIME_TO_STRING(_anyTime^);
  
ELSIF data.TypeClass = __SYSTEM.TYPE_CLASS.TYPE_STRING THEN
  _anyString := data.pValue;
  AnyToString := _anyString^;
  
ELSIF data.TypeClass = __SYSTEM.TYPE_CLASS.TYPE_WSTRING THEN
  _anyWString := data.pValue;
  _wString := _anyWString^;
  Tc2_Utilities.WSTRING_TO_STRING2(ADR(_string), ADR(_wString), SIZEOF(_wString));
  AnyToString := _string;
  
ELSIF data.TypeClass = __SYSTEM.TYPE_CLASS.TYPE_TIMEOFDAY THEN
  _anyTOD := data.pValue;
  AnyToString := TOD_TO_STRING(_anyTOD^);
  
ELSE
  AnyToString := TO_STRING(data.pValue^);
END_IF

END_FUNCTION

// ---- Utils/DynamicStringBuffer.TcPOU
{attribute 'no_explicit_call' := 'This FB is a CLASS and must be accessed using methods or properties'}
{attribute 'hide_all_locals'}
FUNCTION_BLOCK INTERNAL DynamicStringBuffer
VAR_OUTPUT
	Error : Error; // Error information of this FB
END_VAR
VAR
	_fifo : Tc2_Utilities.FB_StringRingBuffer; // Necessary to buffer log data until it has been written to file.
	_memoryManager : Tc3_DynamicMemory.FB_DynMem_Manager; // Memory manager, required by DynMem_Buffer.
	_dynamicMemoryBuffer : Tc3_DynamicMemory.FB_DynMem_Buffer(ipMemMan := _memoryManager); // Provides dynamic buffer for Fifo. Is extended automatically if more than the
																   // default buffer size is needed.                  
	_busy : BOOL; // Buffer is busy; typically with writing data to the file system.
END_VAR

METHOD AddLine : BOOL
VAR_INPUT
  text : Tc2_System.T_MaxString; // Text to be added to the buffer
END_VAR
ResizeFifoBufferIfNecessary();
_fifo.A_AddTail(putValue := Tc2_Standard.CONCAT(Tc2_Standard.LEFT(text, 254), '$N'));
END_METHOD

METHOD AddString : BOOL
VAR_INPUT
  text : Tc2_System.T_MaxString; // String to be added to the buffer
END_VAR
ResizeFifoBufferIfNecessary();
_fifo.A_AddTail(putValue := text);
END_METHOD

METHOD PRIVATE AllocateBuffer : BOOL // Allocates buffer FOR the fifo.
VAR_INPUT
  bufferSize : UDINT; // Initial buffer size in BYTEs for fifo buffer.
END_VAR
_dynamicMemoryBuffer.CreateBuffer(nSize:=bufferSize, bReset:=TRUE);
_fifo.pBuffer := _dynamicMemoryBuffer.pBuffer;
_fifo.cbBuffer := bufferSize;
END_METHOD

{attribute 'monitoring':='call'}
PROPERTY Busy : BOOL
GET
Busy := _busy;
END_GET
SET // PRIVATE
_busy := Busy;
END_SET
END_PROPERTY

METHOD FB_exit : BOOL
VAR_INPUT
  bInCopyCode : BOOL; // if TRUE, the exit method is called for exiting an instance that is copied afterwards (online change).
END_VAR
_dynamicMemoryBuffer.Clear();
END_METHOD

METHOD FlushCache : BOOL
_fifo.A_Reset();
END_METHOD

METHOD INTERNAL Init : BOOL
VAR_INPUT
	bufferSize : UDINT; // Initial buffer size in BYTEs for fifo buffer.
END_VAR
AllocateBuffer(bufferSize);
END_METHOD

{attribute 'hide_all_locals'}
METHOD PersistToFile : BOOL
VAR_INPUT
  enable: BOOL; // TRUE starts persistence mechanism
  fileName : Tc2_System.T_MaxString; // File name including its path
END_VAR
VAR_INST
  state : PersistToFileState;
  
  fileOpen : Tc2_System.FB_FileOpen;
  fileHandle : UINT;
  
  fileWrite : Tc2_System.FB_FileWrite;
  lockFileWriteToForceRisingEdge : BOOL; // filePuts can only be executed every other cycle
                                         // since it needs a rising edge to execute.
  fileClose : Tc2_System.FB_FileClose;
  
  buffer : ARRAY[0..CONSTANTS.BufferSize] OF BYTE;
  currentBufferPos : UDINT;
  fifoHeadString : Tc2_System.T_MaxString;
  fifoHeadLength : UDINT;
  fifoHeadBytes : ARRAY[0..Tc2_System.MAX_STRING_LENGTH] OF BYTE;
  i : UINT;
END_VAR
VAR CONSTANT
  NetId : STRING := '';
  Timeout : TIME := DEFAULT_ADS_TIMEOUT;
  MaxLogsPerCycle : UINT := UDINT_TO_UINT(CONSTANTS.BufferSize / Tc2_System.MAX_STRING_LENGTH);
  MaxBufferPosition : UDINT := (SIZEOF(buffer)-Tc2_System.MAX_STRING_LENGTH);
END_VAR
// State machine
// Using if-statements instead of case for performance reasons:
// Some states execute instantly and allow thus the next state 
// to start within the same plc cycle.

// *** I D L E ***
IF state = PersistToFileState.Idle THEN
  lockFileWriteToForceRisingEdge := FALSE;
  IF _fifo.nCount > 0 AND enable THEN 
    lockFileWriteToForceRisingEdge := FALSE;
    state := PersistToFileState.OpenFile;
  END_IF
END_IF
    
// *** O P E N   F I L E ***
fileOpen(sNetId := NetId, sPathName := fileName, nMode := FOPEN_MODEAPPEND OR FOPEN_MODETEXT, 
           ePath := PATH_GENERIC, bExecute := (state = PersistToFileState.OpenFile), tTimeout := Timeout,
           hFile => fileHandle);

IF state = PersistToFileState.OpenFile THEN
  IF fileOpen.bError THEN
    state := PersistToFileState.CloseFile;
  ELSIF NOT fileOpen.bBusy THEN
    state := PersistToFileState.GetStringFromFifo; 
  END_IF
END_IF 

// *** P O P   F R O M   F I F O ***
IF state = PersistToFileState.GetStringFromFifo THEN
  IF NOT lockFileWriteToForceRisingEdge THEN
    currentBufferPos := 0;
    FOR i:=0 TO MaxLogsPerCycle DO
      IF _fifo.nCount <= 0 THEN EXIT; END_IF
      IF currentBufferPos >= MaxBufferPosition THEN EXIT; END_IF
      
      _fifo.A_RemoveHead(getValue => fifoHeadString); 
      fifoHeadBytes := MAXSTRING_TO_BYTEARR(fifoHeadString);
      fifoHeadLength := INT_TO_UDINT(LEN(fifoHeadString));
      MEMCPY(
        destAddr  :=  ADR(buffer) + SIZEOF(BYTE) * currentBufferPos,
        srcAddr   :=  ADR(fifoHeadBytes),
        n     :=  fifoHeadLength);    
      currentBufferPos := currentBufferPos + fifoHeadLength;  
    END_FOR
    state := PersistToFileState.AppendDataToFile;
  END_IF
  lockFileWriteToForceRisingEdge := FALSE;
END_IF
  
// *** W R I T E   T O   F I L E ***
fileWrite(
  sNetId := NetId, 
  hFile := fileHandle, 
  pWriteBuff := ADR(buffer),
  cbWriteLen := currentBufferPos,
  bExecute := state = PersistToFileState.AppendDataToFile, 
  tTimeout := Timeout); 

IF state = PersistToFileState.AppendDataToFile THEN
  lockFileWriteToForceRisingEdge := TRUE;   
  IF fileWrite.bError THEN
    state := PersistToFileState.CloseFile;
  ELSIF _fifo.nCount > 0 AND NOT fileWrite.bBusy THEN
    state := PersistToFileState.GetStringFromFifo; 
  ELSIF _fifo.nCount = 0 THEN
    state := PersistToFileState.CloseFile;
  END_IF
END_IF
    
// *** C L O S E   F I L E ***
fileClose(
  sNetId := NetId, hFile := fileHandle, 
  bExecute := (state = PersistToFileState.CloseFile), tTimeout := Timeout);

IF state = PersistToFileState.CloseFile THEN
  IF NOT fileClose.bBusy THEN state := PersistToFileState.Idle; END_IF
END_IF

// Close file in case of error
IF fileOpen.bError THEN state := PersistToFileState.CloseFile; END_IF
IF fileWrite.bError THEN state := PersistToFileState.CloseFile; END_IF
IF NOT _fifo.bOk AND _fifo.nCount > 0 AND state <> PersistToFileState.Idle THEN 
  state := PersistToFileState.CloseFile; 
END_IF

// Error handling
IF fileOpen.bError THEN
  Error.Active := TRUE;
  Error.Code := ErrorCodes.OpeningFileFailed;
  Error.Info := Tc2_Standard.CONCAT('Opening file failed. Error thrown by FB_FileOpen. Consult Beckhoff InfoSys. Internal Error: ', UDINT_TO_STRING(fileOpen.nErrId));
ELSIF fileWrite.bError THEN
  Error.Active := TRUE;
  Error.Code := ErrorCodes.WritingToFileFailed;
  Error.Info := Tc2_Standard.CONCAT('Writing to file failed. Error thrown by FB_FileWrite. Consult Beckhoff InfoSys. Internal Error: ', UDINT_TO_STRING(fileWrite.nErrId));
ELSIF fileClose.bError THEN
  Error.Active := TRUE;
  Error.Code := ErrorCodes.ClosingFileFailed;
  Error.Info := Tc2_Standard.CONCAT('Closing file failed. Error thrown by FB_FileClose. Consult Beckhoff InfoSys. Internal Error: ', UDINT_TO_STRING(fileClose.nErrId));
ELSIF NOT _fifo.bOk AND _fifo.nCount > 0 THEN
  Error.Active := TRUE;
  Error.Code := ErrorCodes.FifoOverflow;
  Error.Info := 'FIFO overflow. Check if plc has enough free memory.';
ELSE
  Error.Active := FALSE;
  Error.Code := ErrorCodes.None;
  Error.Info := '';
END_IF

// Set busy state
Busy := (state <> PersistToFileState.Idle OR _fifo.nCount > 0);

(* Uncomment for cyclic logging of state machine, buffer usage & errors

ADSLOGSTR(ADSLOG_MSGTYPE_LOG, 
  Tc2_Standard.CONCAT('****DynamicStringBuffer.state:', 
  Tc2_Standard.CONCAT(UINT_TO_STRING(state),
  Tc2_Standard.CONCAT(', DynamicStringBuffer.hFile:', UINT_TO_STRING(hFile)))), '');

ADSLOGSTR(ADSLOG_MSGTYPE_LOG, 
  Tc2_Standard.CONCAT('****Fifo: used ', 
  Tc2_Standard.CONCAT(UDINT_TO_STRING(Fifo.cbSize),
  Tc2_Standard.CONCAT(' of ', UDINT_TO_STRING(Fifo.cbBuffer)))), '');
  
IF Error.Active THEN
  ADSLOGSTR(ADSLOG_MSGTYPE_LOG, 
    Tc2_Standard.CONCAT('****DynamicStringBuffer.Error: ', Error.Info), 
    '');  
END_IF
*)
END_METHOD

METHOD PopHead : Tc2_System.T_MaxString
VAR_INST
  headString : Tc2_System.T_MaxString;
END_VAR
_fifo.A_RemoveHead(getValue => headString);
PopHead := headString;
END_METHOD

// Resizes the buffer for the FIFO if necessary
METHOD PRIVATE ResizeFifoBufferIfNecessary : BOOL
VAR
  requiredSize : UDINT;
  newSize : DINT;
END_VAR
requiredSize := _fifo.cbSize + (Tc2_System.MAX_STRING_LENGTH + Constants.FifoOverhead);

IF requiredSize > _fifo.cbBuffer THEN
  _dynamicMemoryBuffer.Resize(nSize := requiredSize*SIZEOF(BYTE), bPreserve:=TRUE, bReset:=TRUE);
  _fifo.pBuffer := _dynamicMemoryBuffer.pBuffer;
  _fifo.cbBuffer := requiredSize;
END_IF
END_METHOD

END_FUNCTION_BLOCK

// ---- Utils/DateTime.TcPOU
/// Generate time data in different formats.
{attribute 'no_explicit_call' := 'This FB is a CLASS and must be accessed using methods or properties'}
{attribute: 'hide_all_locals'}
FUNCTION_BLOCK DateTime
VAR
	local_system_time : Tc2_Utilities.FB_LocalSystemTime;
	get_system_time : Tc2_System.GetSystemTime;
	time_zone_info : Tc2_Utilities.FB_GetTimeZoneInformation;
	local_time : Tc2_Utilities.FB_SystemTimeToTzSpecificLocalTime;
	local_system_time_valid : Tc2_Standard.R_Trig;
	utc_time : Tc2_Utilities.FB_TzSpecificLocalTimeToFileTime;
END_VAR

/// Returns local time as `Tc2_Utilities.T_FileTime`.
{attribute 'monitoring':='variable'}
PROPERTY AsLocalFileTime : Tc2_Utilities.T_FileTime
GET
AsLocalFileTime := SYSTEMTIME_TO_FILETIME(THIS^.AsLocalSystemTime);
END_GET
END_PROPERTY

/// Returns local time as `Tc2_Utilities.TimeStruct`.
{attribute 'monitoring':='variable'}
PROPERTY AsLocalSystemTime : Tc2_Utilities.TimeStruct
GET
AsLocalSystemTime := local_system_time.systemTime;
END_GET
END_PROPERTY

/// Returns local time as string.
{attribute 'monitoring':='variable'}
PROPERTY AsLocalSystemTimeString : Tc2_System.T_MaxString
GET
AsLocalSystemTimeString := Tc2_Utilities.SystemTime_To_String(THIS^.AsLocalSystemTime);
END_GET
END_PROPERTY

/// Returns UTC time as `Tc2_Utilities.T_FileTime`.
{attribute 'monitoring':='variable'}
PROPERTY AsUtcFileTime : Tc2_Utilities.T_FileTime
GET
AsUtcFileTime := utc_time.out;
END_GET
END_PROPERTY

METHOD CyclicCall
// Get local system time
local_system_time(
	sNetID  :=  '',
	bEnable :=  TRUE,
	dwCycle :=  1,
	dwOpt :=  1,
	tTimeout:=  DEFAULT_ADS_TIMEOUT
);

// Get timezone information
time_zone_info(
	sNetID := '',
	bExecute := TRUE,
	tTimeout := DEFAULT_ADS_TIMEOUT
);

// Convert local time to utc time
utc_time(
	in := THIS^.AsLocalFileTime,
	tzInfo := time_zone_info.tzInfo
);
 
// Finished retrieving time data
local_system_time_valid(Clk := local_system_time.bValid);
END_METHOD

/// When calling `DateTime` the first time, it takes some time until all time and timezone information is available.
/// `Done` is `TRUE` for one cycle, once all the data is ready. 
{attribute 'monitoring':='call'}
PROPERTY Done : BOOL
GET
Done := local_system_time_valid.Q;
END_GET
END_PROPERTY

// Replaces placeholders in format string by the actual time values.
{attribute 'hide_all_locals'}
{attribute 'hide'}
METHOD PRIVATE ReplaceFormatPlaceholder : STRING
VAR_INPUT
	format : STRING;
	length : INT;
	time_type : STRING(1);
END_VAR
VAR_INST
	i : INT;
	replace_string : STRING;
	time_string : STRING;
END_VAR
VAR
	local_system_time : Tc2_Utilities.TimeStruct;
END_VAR
local_system_time := THIS^.AsLocalSystemTime;

IF    time_type = 'Y' THEN time_string := TO_STRING(local_system_time.wYear);
ELSIF time_type = 'M' THEN time_string := TO_STRING(local_system_time.wMonth);
ELSIF time_type = 'D' THEN time_string := TO_STRING(local_system_time.wDay);
ELSIF time_type = 'h' THEN time_string := TO_STRING(local_system_time.wHour);
ELSIF time_type = 'm' THEN time_string := TO_STRING(local_system_time.wMinute);
ELSIF time_type = 's' THEN time_string := TO_STRING(local_system_time.wSecond);
ELSIF time_type = 'i' THEN time_string := TO_STRING(local_system_time.wMilliseconds);
ELSE
	time_string := '';
END_IF

replace_string := '';

IF length > Tc2_Standard.Len(time_string) THEN
	FOR i:=1 TO length - Tc2_Standard.Len(time_string) DO
		replace_string := Tc2_Standard.Concat(replace_string, '0');
	END_FOR
	replace_string := Tc2_Standard.Concat(replace_string, time_string);
ELSE
	replace_string := Tc2_Standard.Right(time_string, length);
END_IF

ReplaceFormatPlaceholder := Tc2_Standard.Replace(format, replace_string, length, Tc2_Standard.Find(format, time_type));
END_METHOD

/// Returns a formatted string containing the actual time information 
/// - `Y` : year
/// - `M` : month
/// - `D` : day
/// - `h` : hour 
/// - `m` : minute
/// - `s` : second
/// - `i` : millisecond
/// 
/// Example:    
/// _YYMMDD-hh:mm:ss:iii_   
/// => _20210812-12:30:22:123_
{attribute 'hide_all_locals'}
METHOD PUBLIC ToFormatString : Tc2_System.T_MaxString
VAR_INPUT
  /// Format the timestamp should have.
  format : STRING;
END_VAR
VAR_INST
  inputString : STRING;
  c : STRING(1);
  formattedString : Tc2_System.T_MaxString;
END_VAR
VAR
  year : INT := 0;
  month : INT := 0;
  day : INT := 0;
  hour : INT := 0;
  minute : INT := 0;
  second : INT := 0;
  millisecond : INT := 0;
END_VAR
VAR CONSTANT
  ValidFormat : STRING := 'YMDhms';
END_VAR
// Parses "format" and returns a adequatly formatted string containing the time information
inputString := format;

WHILE Tc2_Standard.LEN(inputString) > 0 DO
  c := Tc2_Standard.LEFT(inputString, 1);
  
  IF    c = 'Y' THEN year := year + 1;
  ELSIF c = 'M' THEN month := month + 1;
  ELSIF c = 'D' THEN day := day + 1;
  ELSIF c = 'h' THEN hour := hour + 1;
  ELSIF c = 'm' THEN minute := minute + 1;
  ELSIF c = 's' THEN second := second + 1;
  ELSIF c = 'i' THEN millisecond := millisecond + 1;
  END_IF
  
  inputString := Tc2_Standard.DELETE(inputString, 1, 1);
END_WHILE

formattedString := ReplaceFormatPlaceholder(format, year, 'Y');
formattedString := ReplaceFormatPlaceholder(formattedString, month, 'M');
formattedString := ReplaceFormatPlaceholder(formattedString, day, 'D');
formattedString := ReplaceFormatPlaceholder(formattedString, hour, 'h');
formattedString := ReplaceFormatPlaceholder(formattedString, minute, 'm');
formattedString := ReplaceFormatPlaceholder(formattedString, second, 's');
formattedString := ReplaceFormatPlaceholder(formattedString, millisecond, 'i');

ToFormatString := formattedString;
END_METHOD

END_FUNCTION_BLOCK

// ---- Logger/TcLogCore.TcPOU
/// `TcLogCore` provides the base functionality of the logger and sets the configuration.
/// The logger can be configured by calling its methods that set the configuration.
///
/// > [!NOTE]
/// > `TcLogCore.RunLogger()` should be called once each cycle. The configuration methods should be called **before** 
/// > `RunLogger` is called.
///
/// When declaring an instance of TcLogCore, the ininital buffer size has to be set. If the buffer size is set too low, it will expand
/// automatically if enough memory is available.
///
/// To set the inital buffer size to accomodate 100 messages, use it like this:
///
/// ```st
/// VAR
///   my_logger: TcLogCore(BufferSize := 100 * (Tc2_System.MAX_STRING_LENGTH * Constants.FifoOverhead));
/// END_VAR
/// ```
///
{attribute 'linkalways'}
{attribute 'no_explicit_call' := 'This FB is a CLASS and must be accessed using methods or properties'}
//{attribute 'hide_all_locals'}
FUNCTION_BLOCK PUBLIC TcLogCore IMPLEMENTS ILogCore
VAR
	logging_singleton : TcLog; // Logger-Singleton: Required to provide Singleton-functionality for TcLog.
	utc_time_as_file_time : Tc2_Utilities.T_FileTime; // Current utc time as filetime
	local_time_as_system_time : Tc2_Utilities.TimeStruct; // Current local time as timestring
	local_time_as_string : STRING; // Current local time as string
	log_cache : DynamicStringBuffer; // Dynamic string buffer to cache logs to be processed
	start_logging_configuration : BOOL; // Aux variable to provide fluent interface.
	internal_error_occured : BOOL; // Aux variable to log internal errors to Error-property.                                                   				
	_config : LoggingConfiguration := (
		MinimumLevel := LogLevel.Debug,
		Delimiter := '|',
		IncludeInstancePath := FALSE,
		TimestampFormat := 'YYYYMMDD_hhmm_',
		ValidTimestampsOnly := FALSE
	); // Logging configuration. Is set by invoking configuration methods.
	_error : Error; // Contains information about internal error.
	_busy : BOOL; // Logger is busy, typically with writing logs to the file system.
	time_info_ready : BOOL := FALSE; // Set to true once the time information is available
	
	default_log_target_adapter : AdsLogTargetAdapter;

	adapter_1 : LogTargetAdapter := default_log_target_adapter;
	adapter_2 : LogTargetAdapter;
	adapter_3 : LogTargetAdapter;
END_VAR

// Nothing to be done here. Logger works by invoking its methods.
// "RunLogger" contains all the implementation that has to be processed cyclically.

METHOD PUBLIC AddAdapter1 : REFERENCE TO TcLogCore
VAR_INPUT
	adapter : LogTargetAdapter;
END_VAR
IF adapter <> 0 THEN
	adapter_1 := adapter;
END_IF

AddAdapter1 REF= THIS^;
END_METHOD

METHOD PUBLIC AddAdapter2 : REFERENCE TO TcLogCore
VAR_INPUT
	adapter : LogTargetAdapter;
END_VAR
IF adapter <> 0 THEN
	adapter_2 := adapter;
END_IF

AddAdapter2 REF= THIS^;
END_METHOD

METHOD PUBLIC AddAdapter3 : REFERENCE TO TcLogCore
VAR_INPUT
	adapter : LogTargetAdapter;
END_VAR
IF adapter <> 0 THEN
	adapter_3 := adapter;
END_IF

AddAdapter3 REF= THIS^;
END_METHOD

/// `Busy` evaluates to `TRUE` as long as the log file is kept open to append new log messages
/// or there are pending messages in the queue to be written to the logfile.
{attribute 'monitoring':='call'}
PROPERTY PUBLIC Busy : BOOL
GET // PUBLIC
Busy := _busy;
END_GET
SET // PRIVATE
_busy := Busy;
END_SET
END_PROPERTY

/// Returns the current configuration of the logger.
{attribute 'monitoring':='variable'}
PROPERTY PUBLIC Configuration : LoggingConfiguration
GET // PUBLIC
Configuration := _config;
END_GET
END_PROPERTY

/// Returns information about internal errors.
{attribute 'monitoring':='call'}
{attribute 'suppress_wrn_C0410'}
PROPERTY Error : REFERENCE TO Error
GET
Error REF= _error;
END_GET
END_PROPERTY

METHOD FB_init : BOOL
VAR_INPUT
	bInitRetains : BOOL; // if TRUE, the retain variables are initialized (warm start / cold start)
	bInCopyCode : BOOL; // if TRUE, the instance afterwards gets moved into the copy code (online change)
	/// Initial buffer size for the internal log message buffer
	bufferSize : UDINT;
END_VAR
logging_singleton.Init(THIS^);
log_cache.Init(bufferSize);
END_METHOD

/// Configuration method. If this method is called, the instance path where the log 
/// messages has been triggered will be included in the log message. 
METHOD PUBLIC IncludeInstancePath : REFERENCE TO TcLogCore
_config.IncludeInstancePath := TRUE;

IncludeInstancePath REF= This^;
END_METHOD

/// Logger method. It should only be called from within objects that implement `ILog`.
/// Logs in the standard format. This includes
/// - timestamp
/// - log level
/// - log message
/// - instance path of logging source (optional)
/// The message will only be logged if the logging level exceeds the configured minimum logging level.
METHOD PUBLIC LogStandardFormat : BOOL
VAR_INPUT
	/// Instance path of calling logger to locate source of logging message.
	instance_path : Tc2_System.T_MaxString;

	/// Log level of message. 
	level : LogLevel; 

	/// Data to be logged.
	message : Tc2_System.T_MaxString;	
END_VAR
VAR_INST
	event : LogEvent;
END_VAR
IF level >= _config.MinimumLevel AND (TimeInfoReady OR NOT _config.ValidTimestampsOnly) THEN
	event.timestamp := local_time_as_system_time;
	event.level := level;
	event.logger := instance_path;
	event.message := message;

	IF adapter_1 <> 0 THEN
		adapter_1.SendLogEvent(event);
	END_IF
	
	IF adapter_2 <> 0 THEN
		adapter_2.SendLogEvent(event);
	END_IF
	
	IF adapter_3 <> 0 THEN
		adapter_3.SendLogEvent(event);
	END_IF
END_IF
END_METHOD

/// Configuration method.
/// Sets the minimum log level. Log messages below this level 
/// will not be logged.
METHOD PUBLIC MinimumLevel : REFERENCE TO TcLogCore
VAR_INPUT
  /// Minimum log level to be logged.
	level : LogLevel; 
END_VAR
_config.MinimumLevel := level;

MinimumLevel REF=THIS^;
END_METHOD

/// Cyclic method of Logger.
/// This method has to be executed in every PLC cycle and runs 
/// all internal methods that have to be executed cyclically.
/// > [!NOTE]
/// > This method should be the last method of `TcLogCore` to be called in each cycle.
{attribute 'hide_all_locals'}
METHOD PUBLIC RunLogger : BOOL
VAR_INST
	new_day : Tc2_Standard.R_Trig; 
	date_time : DateTime;
	delete_expired_log_files : DeleteOldFiles;
	file_name_string_builder : StringBuilder;
	time_stamp : STRING; // Timestamp used for filename
END_VAR
// Generate time data (shared state)
date_time.CyclicCall();
IF date_time.Done THEN
	time_info_ready := TRUE;
END_IF

local_time_as_system_time := date_time.AsLocalSystemTime;
local_time_as_string := date_time.AsLocalSystemTimeString;
utc_time_as_file_time := date_time.AsUtcFileTime;

IF adapter_1 <> 0 THEN
	adapter_1.Run();
END_IF

IF adapter_2 <> 0 THEN
	adapter_2.Run();
END_IF

IF adapter_3 <> 0 THEN
	adapter_3.Run();
END_IF

// Reset Logging configuration: neccesary in order to provide fluent interface
start_logging_configuration := FALSE;
END_METHOD

/// Configuration method
/// Sets delimiter between different columns of log file.
METHOD PUBLIC SetDelimiter : REFERENCE TO TcLogCore
VAR_INPUT
  /// Delimiter between different columns of log file.
	delimiter : STRING(1); 
END_VAR
_config.Delimiter := delimiter;

SetDelimiter REF=THIS^;
END_METHOD

/// `TimeInfoReady` evaluates to `TRUE` once the time information used by determine
/// the timestamp for the message is available.
{attribute 'monitoring':='call'}
PROPERTY PUBLIC TimeInfoReady : BOOL
GET // PUBLIC
TimeInfoReady := time_info_ready;
END_GET
END_PROPERTY

/// Configuration method.
/// Sets the format of the timestamp in the file name. 
/// 
/// The following format options are available:
///	Y : year
///	M : month
/// D : day
/// h : hour 
/// m : minute
/// s : second
/// i : millisecond
/// 
/// Example: _YYMMDD-hh:mm:ss:iii_
/// => _20210812-12:30:22:123_
METHOD PUBLIC TimestampFormat : REFERENCE TO TcLogCore
VAR_INPUT
  /// Format the timestamp should have.
	format : STRING; 
END_VAR
_config.TimestampFormat := format;

TimestampFormat REF= THIS^;
END_METHOD

/// Configuration method. If this method is called, only valid timestamps are logged.
/// Note that using this configuration will skip logging anything during the first few PLC cycles, 
/// as TwinCAT needs a few cycles to initialize its time information.
METHOD PUBLIC ValidTimestampsOnly : REFERENCE TO TcLogCore
_config.ValidTimestampsOnly := TRUE;

ValidTimestampsOnly REF= This^;
END_METHOD

END_FUNCTION_BLOCK

// ---- Logger/TcLogTrig.TcPOU
/// This function block can be used to log on rising or falling edges.
/// For each signal that should be watched, a separate instance of `TcLogTrig` 
/// must be created.
{attribute 'linkalways'}
{attribute 'no_explicit_call' := 'This FB is a CLASS and must be accessed using methods or properties'}
FUNCTION_BLOCK PUBLIC TcLogTrig EXTENDS TcLog

/// Logs data on falling edge of `CLK`.
{attribute 'hide_all_locals'}
METHOD PUBLIC OnFallingEdge : REFERENCE TO TcLog
VAR_INPUT
  /// Falling edge triggers logging the data.
  CLK : BOOL; 
END_VAR
VAR_INST
    fTrig : Tc2_Standard.F_TRIG;
END_VAR
fTrig(CLK:=CLK);

SUPER^.OnCondition(fTrig.Q);

OnFallingEdge REF= THIS^;
END_METHOD

/// Logs data on rising edge of `CLK`.
{attribute 'hide_all_locals'}
METHOD PUBLIC OnRisingEdge : REFERENCE TO TcLog
VAR_INPUT
  /// Rising edge logs data.
  CLK : BOOL; 
END_VAR
VAR_INST
    rTrig : Tc2_Standard.R_TRIG;
END_VAR
rTrig(CLK:=CLK);

SUPER^.OnCondition(rTrig.Q);

OnRisingEdge REF= THIS^;
END_METHOD

END_FUNCTION_BLOCK

// ---- Utils/GetFileAgeInSeconds.TcPOU
{attribute 'hide'}
FUNCTION INTERNAL GetFileAgeInSeconds : DINT
VAR_INPUT
  currentUtcTime : Tc2_Utilities.T_FILETIME;
  findFileEntry : Tc2_Utilities.ST_FindFileEntry;
END_VAR
VAR
  _timeLastWriteAccess : Tc2_Utilities.T_ULARGE_INTEGER;
  _fileTimeAsULINT : Tc2_Utilities.T_ULARGE_INTEGER;
  _fileTimeDifference : Tc2_Utilities.T_ULARGE_INTEGER;
END_VAR
VAR CONSTANT
  OneSecondInOneHundredNanoSecondsIntervals : LREAL := 1000*1000*10;
END_VAR

// Local file time
_fileTimeAsULINT.dwLowPart := currentUtcTime.dwLowDateTime;
_fileTimeAsULINT.dwHighPart := currentUtcTime.dwHighDateTime;

// Write access is UTC
_timeLastWriteAccess.dwLowPart := findFileEntry.lastWriteTime.dwLowDateTime;
_timeLastWriteAccess.dwHighPart := findFileEntry.lastWriteTime.dwHighDateTime;
_fileTimeDifference := UInt64Sub64(_fileTimeAsULINT, _timeLastWriteAccess);

GetFileAgeInSeconds := LREAL_TO_DINT(UINT64_TO_LREAL(_fileTimeDifference)/(OneSecondInOneHundredNanoSecondsIntervals));

END_FUNCTION
